# EPICS autosave request: softGlueApp/Db/softGlue_SignalShow_settings.req
$(P)$(H)ReadRate.SCAN
